{attribute 'GeneratedUsingTerminal: EL2202-0000-0016'}
{attribute addProperty BoxType "EL2202-0000-0016"}
{attribute addProperty Id "Channel_1AT %Q*Channel_54BE63B32Channel_2AT %Q*Channel_54BE63B32WcStateAT %I*WcState_0B2B16F91InfoDataAT %I*InfoData_6F19DB2B2"}
{attribute addProperty CRC "3838898774"}
{attribute addProperty Size "7"}
TYPE EL2202_E4D0F256 EXTENDS EtcSlaveTerminalBase_947E5A46 :
STRUCT
	{attribute addProperty Name "Channel_1"}
	Channel_1 : Channel_54BE63B3;
	{attribute addProperty Name "Channel_2"}
	Channel_2 : Channel_54BE63B3;
	{attribute addProperty Name "WcState"}
	WcState : WcState_0B2B16F9;
	{attribute addProperty Name "InfoData"}
	InfoData : InfoData_6F19DB2B;
END_STRUCT
END_TYPE

(* stored: Version 1.2.0.0, ProductVersion 3.1.4024.9
   DUT EL2202_E4D0F256: Id {5d9ea262-9fa6-4155-84a6-4b564bca2a72} *)
